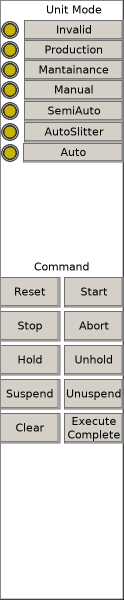
VISUALIZATION VIS_TemplateCommand  // 124x600
VAR_IN_OUT
	eModeCommand	: DINT;
	eStateCommand	: DINT;
	eModeStatus		: DINT;
	eStateStatus	: DINT;
	bModeChangeReq	: BOOL;
END_VAR
    Rectangle (0,0 124x600)
    Lamp1 (0,20 20x20), variable: (eModeStatus = 0), style: Lamp-Lamp1-Yellow
    Button (24,20 100x20), "Invalid", colour toggle: (eModeStatus = 0)
        tap bModeChangeReq
        OnMouseClick: execute { eModeCommand := 0; }
    Lamp1 (0,40 20x20), variable: (eModeStatus = 1), style: Lamp-Lamp1-Yellow
    Button (24,40 100x20), "Production"
        tap bModeChangeReq
        OnMouseClick: execute { eModeCommand := 1; }
    Lamp1 (0,60 20x20), variable: (eModeStatus = 2), style: Lamp-Lamp1-Yellow
    Button (24,60 100x20), "Mantainance"
        tap bModeChangeReq
        OnMouseClick: execute { eModeCommand := 2; }
    Lamp1 (0,80 20x20), variable: (eModeStatus = 3), style: Lamp-Lamp1-Yellow
    Button (24,80 100x20), "Manual"
        tap bModeChangeReq
        OnMouseClick: execute { eModeCommand := 3; }
    Button (0,277 60x30), "Reset"
        OnMouseClick: execute { eStateCommand := 1; }
    Button (64,277 60x30), "Start"
        OnMouseClick: execute { eStateCommand := 2; }
    Button (0,311 60x30), "Stop"
        OnMouseClick: execute { eStateCommand := 3; }
    Button (0,345 60x30), "Hold"
        OnMouseClick: execute { eStateCommand := 4; }
    Button (64,345 60x30), "Unhold"
        OnMouseClick: execute { eStateCommand := 5; }
    Button (0,379 60x30), "Suspend"
        OnMouseClick: execute { eStateCommand := 6; }
    Button (64,379 60x30), "Unuspend"
        OnMouseClick: execute { eStateCommand := 7; }
    Button (0,413 60x30), "Clear"
        OnMouseClick: execute { eStateCommand := 9; }
    Label (0,257 124x20), "Command"
    Button (64,311 60x30), "Abort"
        OnMouseClick: execute { eStateCommand := 8; }
    Button (64,413 60x30), "Execute Complete"
        OnMouseClick: execute { MAIN.bExecuteComplete := TRUE; }
    Label (24,0 100x20), "Unit Mode"
    Button (24,101 100x20), "SemiAuto"
        tap bModeChangeReq
        OnMouseClick: execute { eModeCommand := 4; }
    Lamp1 (0,101 20x20), variable: (eModeStatus = 4), style: Lamp-Lamp1-Yellow
    Button (24,122 100x20), "AutoSlitter"
        tap bModeChangeReq
        OnMouseClick: execute { eModeCommand := 5; }
    Lamp1 (0,122 20x20), variable: (eModeStatus = 5), style: Lamp-Lamp1-Yellow
    Button (23,143 101x19), "Auto"
        tap bModeChangeReq
        OnMouseClick: execute { eModeCommand := 6; }
    Lamp1 (0,143 20x20), variable: (eModeStatus = 6), style: Lamp-Lamp1-Yellow
END_VISUALIZATION

(* stored: Version 1.1.0.1, ProductVersion 3.1.4024.12
   Visu VIS_TemplateCommand: Id {d7925750-20c5-4482-a15b-9b1c5b9b40e3} *)
